// Mitsubishi GX Works2 project: 실린더응용2   PLC: Q02/Q02H

PROGRAM MAIN
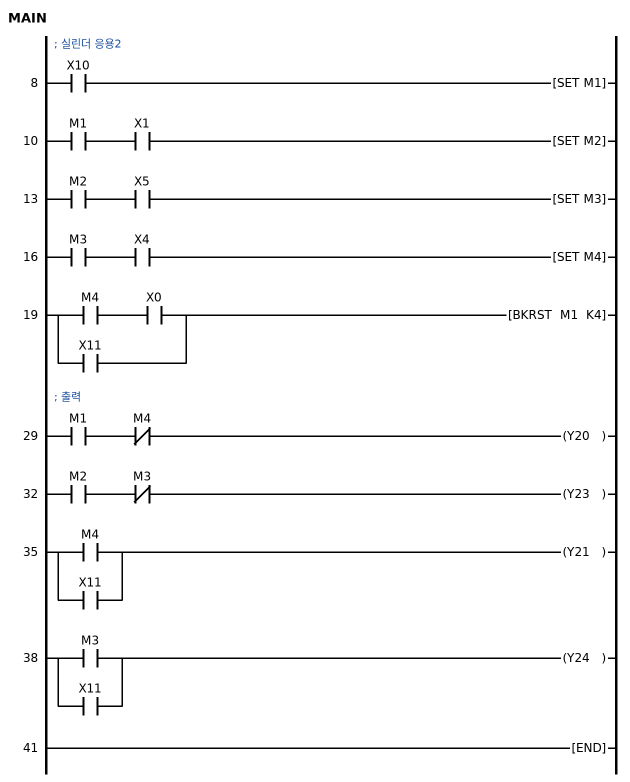
; 실린더 응용2
8     LD      X10
      SET     M1
10    LD      M1
      AND     X1
      SET     M2
13    LD      M2
      AND     X5
      SET     M3
16    LD      M3
      AND     X4
      SET     M4
19    LD      M4
      AND     X0
      OR      X11
      BKRST   M1 K4
; 출력
29    LD      M1
      ANI     M4
      OUT     Y20
32    LD      M2
      ANI     M3
      OUT     Y23
35    LD      M4
      OR      X11
      OUT     Y21
38    LD      M3
      OR      X11
      OUT     Y24
41    END
END_PROGRAM
